% RSLogix 500 project I2P-Job-09 Duncan_Sutton.RSS, saved by version 10.00.00.00 %
PROJECT "ML01A"    % processor: Bul.1763 MicroLogix 1100 Series B %

PROGRAM FILES
  LAD 2   5 rungs

DATA FILES
  O0 OUTPUT  4 elements
  I1 INPUT  6 elements
  S2 STATUS  66 elements
  B3 BINARY  1 elements
  T4 TIMER  1 elements
  C5 COUNTER  1 elements
  R6 CONTROL  1 elements
  N7 INTEGER  1 elements
  F8 FLOAT  1 elements

LADDER 2
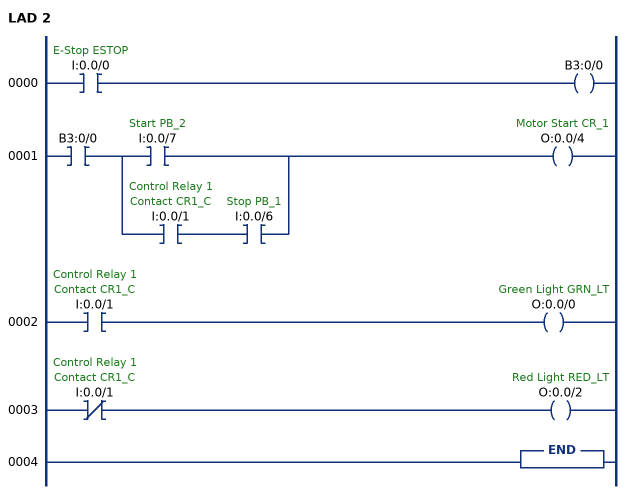
% Rung: 0 %
SOR XIC I:0.0/0 OTE B3:0/0 EOR
%   I:0.0/0  ESTOP  "E-Stop" %
% Rung: 1 %
SOR XIC B3:0/0 BST XIC I:0.0/7 NXB XIC I:0.0/1 XIC I:0.0/6 BND OTE O:0.0/4 EOR
%   I:0.0/7  PB_2  "Start" %
%   I:0.0/1  CR1_C  "Control Relay 1 Contact" %
%   I:0.0/6  PB_1  "Stop" %
%   O:0.0/4  CR_1  "Motor Start" %
% Rung: 2 %
SOR XIC I:0.0/1 OTE O:0.0/0 EOR
%   I:0.0/1  CR1_C  "Control Relay 1 Contact" %
%   O:0.0/0  GRN_LT  "Green Light" %
% Rung: 3 %
SOR XIO I:0.0/1 OTE O:0.0/2 EOR
%   I:0.0/1  CR1_C  "Control Relay 1 Contact" %
%   O:0.0/2  RED_LT  "Red Light" %
% Rung: 4 %
SOR END EOR

OTHER DOCUMENTED ADDRESSES
  I:0.0/2  CR2_C  "Control Relay 2 Contact"
  I:0.0/3  3PSS_PA  "3 Postion Selector Switch Position A"
  I:0.0/4  3PSS_PB  "3 Position Selector Switch Position B"
  I:0.0/5  2PSS_PA  "2 Poistion Selector Switch Position A"
  I:0.0/8  PB_3  "Pushbutton 3"
  O:0.0/1  "Yellow Light"
  O:0.0/3  BLU_LT  "Blue Light"
  O:0.0/5  CR_2  "Control Relay 2"
